{attribute 'GeneratedUsingTerminal: EK1122-0000-0018'}
{attribute addProperty BoxType "EK1122-0000-0018"}
{attribute addProperty Id "Beckhoff_EL2xxxsub_EK1100EK1100_1FC0878B2"}
{attribute addProperty CRC "2521710905"}
{attribute addProperty Size "2"}
TYPE Beckhoff_EL2xxxEK1122_964E4139 EXTENDS EK1122_1FC0878B :
STRUCT
	{attribute addProperty Name "Beckhoff EL2xxxsub EK1100"}
	{attribute addProperty PreviousPort "Beckhoff EL2xxxEK1122 : D"}
	Beckhoff_EL2xxxsub_EK1100 : EK1100_1FC0878B;
END_STRUCT
END_TYPE

(* stored: Version 1.2.0.0, ProductVersion 3.1.4024.9
   DUT Beckhoff_EL2xxxEK1122_964E4139: Id {e43d9ce9-7f98-40a7-8d0c-a76554dbf5f9} *)
